TYPE EL5001_Status :
STRUCT
	{attribute addProperty Name "Data error"}
	DataError : BIT;
	{attribute addProperty Name "Frame error"}
	FrameError : BIT;
	{attribute addProperty Name "Power failure"}
	PowerFailure : BIT;
	{attribute 'hide'}
	{attribute addProperty Name "Bit 4(address x.3)"}
	Bit_4 : BIT;
	{attribute addProperty Name "Bit 5(address x.4)"}
	{attribute 'hide'}
	Bit_5 : BIT;
	{attribute 'hide'}
	{attribute addProperty Name "Bit 6(address x.5)"}
	Bit_6 : BIT;
	{attribute 'hide'}
	{attribute addProperty Name "Bit 7(address x.6)"}
	Bit_7 : BIT;
	{attribute 'hide'}
	{attribute addProperty Name "Bit 8(address x.7)"}
	Bit_8 : BIT;
	{attribute 'hide'}
	{attribute addProperty Name "Bit 9(address x+1.0)"}
	Bit_9 : BIT;
	{attribute 'hide'}
	{attribute addProperty Name "Bit 10(address x+1.1)"}
	Bit_10 : BIT;
	{attribute 'hide'}
	{attribute addProperty Name "Bit 11(address x+1.2)"}
	Bit_11 : BIT;
	{attribute 'hide'}
	{attribute addProperty Name "Bit 12(address x+1.3)"}
	Bit_12 : BIT;
	{attribute 'hide'}
	{attribute addProperty Name "Bit 13(address x+1.4)"}
	Bit_13 : BIT;
	{attribute addProperty Name "Sync error"}
	SyncError : BIT;
	{attribute addProperty Name "TxPDO State"}
	TxPDOState : BIT;
	{attribute addProperty Name "TxPDO Toggle"}
	TxPDOToggle : BIT;
END_STRUCT
END_TYPE

(* stored: Version 1.1.0.1, ProductVersion 3.1.4024.9
   DUT EL5001_Status: Id {f083bcfe-2c16-09ba-21b6-1fb4560e0209} *)
